% RSLogix 500 project rev_pulse_1.6384.RSS, saved by version 8.30.00.16 %
PROJECT "UNTITLED"    % processor: Bul.1763 MicroLogix 1100 Series B %

PROGRAM FILES
  LAD 2   3 rungs

DATA FILES
  O0 OUTPUT  4 elements
  I1 INPUT  6 elements
  S2 STATUS  66 elements
  B3 BINARY  24 elements
  T4 TIMER  1 elements
  C5 COUNTER  1 elements
  R6 CONTROL  1 elements
  N7 INTEGER  2 elements
  F8 FLOAT  10 elements
  L9 MISCELLANY  10 elements

LADDER 2
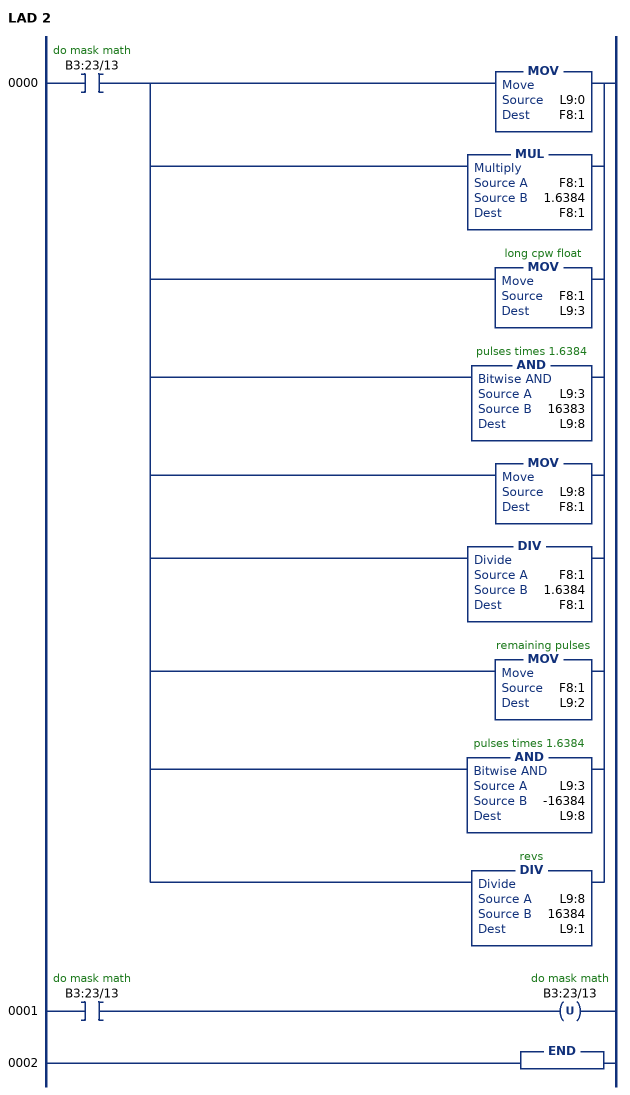
% Rung: 0 %
SOR XIC B3:23/13 BST MOV L9:0 F8:1 NXB MUL F8:1 1.6384 F8:1 NXB MOV F8:1 L9:3 NXB AND L9:3 16383 L9:8 NXB MOV L9:8 F8:1 NXB DIV F8:1 1.6384 F8:1 NXB MOV F8:1 L9:2 NXB AND L9:3 -16384 L9:8 NXB DIV L9:8 16384 L9:1 BND EOR
%   B3:23/13  "do mask math" %
%   L9:0  "long pulse count" %
%   L9:3  "long cpw float" %
%   L9:8  "pulses times 1.6384" %
%   L9:2  "remaining pulses" %
%   L9:1  "revs" %
% Rung: 1 %
SOR XIC B3:23/13 OTU B3:23/13 EOR
%   B3:23/13  "do mask math" %
% Rung: 2 %
SOR END EOR

OTHER DOCUMENTED ADDRESSES
  F8:0  "float rev.pulse"
  L9:4  "long tmp value"
  L9:5  "long exponent"
  L9:6  "misc one bit"
  L9:7  "exponent mask"
  L9:9  "revs times 16k"
  L20:[N7:0]  "current one bit"
  L21:[N7:0]  "current low mask"
  N7:0  "counter 23"
